PROGRAM MAIN
VAR
	a,b,c:INT;
	add1:FB_ADD;
END_VAR

add1(in1:=a , in2:=b , out=>c );

END_PROGRAM

(* stored: Version 1.1.0.1, ProductVersion 3.1.4024.11
   POU MAIN: Id {fd1f92b4-c07e-407e-90a5-b09f217d860b}, SpecialFunc None *)
